INTERFACE I_Room

// sets the temperature, returns the actual status
METHOD M_SetTemperature : BOOL
VAR_INPUT
	bOnOff					: BOOL;
	nTemperature			: REAL;
END_VAR
END_METHOD

// Switches the light on/off with certain illuminance
METHOD M_SwitchLight : BOOL
VAR_INPUT
	bOnOff				: BOOL;
	nIlluminance		: REAL;
END_VAR
END_METHOD

END_INTERFACE

(* stored: Version 1.1.0.1, ProductVersion 3.1.4022.18
   Itf I_Room: Id {d418edf8-67f3-40f7-b4a7-abc90865897d}
   Method M_SetTemperature: Id {a76e8548-9872-43e7-8105-29f65ff90cd4}
   Method M_SwitchLight: Id {f2944ea8-6079-47ea-8650-e69c176afb8e} *)
